FUNCTION_BLOCK fbFuzzyAnd
VAR_INPUT
END_VAR
VAR_OUTPUT
END_VAR
VAR
END_VAR

END_FUNCTION_BLOCK

(* stored: Version 1.1.0.1, ProductVersion 3.1.4024.6
   POU fbFuzzyAnd: Id {fb609b59-bfae-41e3-963c-299cb3a2cec7}, SpecialFunc None *)
